//{{V2}}
DATA_BLOCK DB100

AUTHOR:mh
FAMILY:nb
NAME:nb
VERSION:1.0


       STRUCT
         b0:INT
       b1:INT
       b2:INT
       b3:INT
       b4:INT
       b5:INT
       b6:INT
       b7:INT
       b8:INT
       b9:INT
       END_STRUCT
BEGIN

       b0:=0
       b1:=0
       b2:=0
       b3:=0
       b4:=0
       b5:=0
       b6:=0
       b7:=0
       b8:=0
       b9:=0
END_DATA_BLOCK
